# EPICS substitutions: beckhoffApp/Db/frozen_offsets.substitutions
file "$(TOP)/beckhoffApp/beckhoff_write_pv.template" {
    pattern {P, NAME, PORT, ADSPORT, V, RECTYPE, EPICSDTYP, ADS_TYPE}
    {"\$(P)", "ASTAXES_\$(AXIS_NUM):STCONTROL-FSETPOSITION", "\$(PORT)", "\$(ADSPORT)", "GVL.astAxes[\$(AXIS_NUM)].stControl.fSetPosition", ao, "asynFloat64", "LREAL"}
}
